(* CoDeSys 2.3.9.50 project: test.pr6 *)
(* Libraries: STANDARD.LB6 5.6.98 12:03:02 *)

(* Global variable list: TwinCAT_Import *)
VAR_GLOBAL (* DO NOT CHANGE THIS SHEET MANUALLY! *)
	PlcInVar_0	AT %QB128:	USINT;
	PlcInVar_1	AT %QB129:	USINT;
	PlcInVar_2	AT %QB130:	USINT;
	PlcInVar_3	AT %QB131:	USINT;
	PlcInVar_4	AT %QB132:	USINT;
	PlcInVar_5	AT %QB133:	USINT;
	PlcInVar_6	AT %QB134:	USINT;
	PlcInVar_7	AT %QB135:	USINT;
	PlcInVar_8	AT %QB136:	USINT;
	PlcInVar_9	AT %QB137:	USINT;
	PlcInVar_10	AT %QB138:	USINT;
	PlcInVar_11	AT %QB139:	USINT;
	PlcInVar_12	AT %QB140:	USINT;
	PlcInVar_13	AT %QB141:	USINT;
	PlcInVar_14	AT %QB142:	USINT;
	PlcInVar_15	AT %QB143:	USINT;
	PlcOutVar_0	AT %IB128:	USINT;
	PlcOutVar_1	AT %IB129:	USINT;
	PlcOutVar_2	AT %IB130:	USINT;
	PlcOutVar_3	AT %IB131:	USINT;
	PlcOutVar_4	AT %IB132:	USINT;
	PlcOutVar_5	AT %IB133:	USINT;
	PlcOutVar_6	AT %IB134:	USINT;
	PlcOutVar_7	AT %IB135:	USINT;
	PlcOutVar_8	AT %IB136:	USINT;
	PlcOutVar_9	AT %IB137:	USINT;
	PlcOutVar_10	AT %IB138:	USINT;
	PlcOutVar_11	AT %IB139:	USINT;
	PlcOutVar_12	AT %IB140:	USINT;
	PlcOutVar_13	AT %IB141:	USINT;
	PlcOutVar_14	AT %IB142:	USINT;
	PlcOutVar_15	AT %IB143:	USINT;
	Terminal_2_KL1408_1_Input	AT %IX0.0:	BOOL;
	Terminal_2_KL1408_2_Input	AT %IX0.1:	BOOL;
	Terminal_2_KL1408_3_Input	AT %IX0.2:	BOOL;
	Terminal_2_KL1408_4_Input	AT %IX0.3:	BOOL;
	Terminal_2_KL1408_5_Input	AT %IX0.4:	BOOL;
	Terminal_2_KL1408_6_Input	AT %IX0.5:	BOOL;
	Terminal_2_KL1408_7_Input	AT %IX0.6:	BOOL;
	Terminal_2_KL1408_8_Input	AT %IX0.7:	BOOL;
	Terminal_3_KL2408_1_Output	AT %QX0.0:	BOOL;
	Terminal_3_KL2408_2_Output	AT %QX0.1:	BOOL;
	Terminal_3_KL2408_3_Output	AT %QX0.2:	BOOL;
	Terminal_3_KL2408_4_Output	AT %QX0.3:	BOOL;
	Terminal_3_KL2408_5_Output	AT %QX0.4:	BOOL;
	Terminal_3_KL2408_6_Output	AT %QX0.5:	BOOL;
	Terminal_3_KL2408_7_Output	AT %QX0.6:	BOOL;
	Terminal_3_KL2408_8_Output	AT %QX0.7:	BOOL;
END_VAR

(* POU MAIN, LD *)
PROGRAM MAIN
VAR
	entrada AT %IX0.0:BOOL;
	salida AT %QX0.0:BOOL;
END_VAR
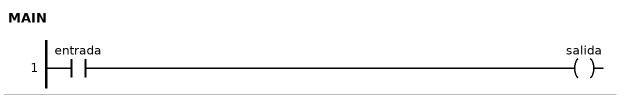
_LD_ (* Ladder Diagram *)
NETWORK 1
	[entrada] --- (salida)
_END_LD_
(* the same logic as Structured Text *)
(* Network 1 *)
salida := entrada;
END_PROGRAM

(* Visualisation Prueba
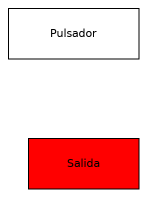
rectangle at (100,70)-(231,121): text "Pulsador"; taps MAIN.entrada
rectangle at (120,200)-(231,251): text "Salida"; alarm colour if MAIN.salida
*)
